TYPE E_Typ_MER_MODE :
(
	/// 0= main mode automatic, controller automatically merge hangers from different lines dependent E_Typ_MER_AUTO_MODE
	Automatic := 0,
	/// 1= main mode on command, in case if merger work as charge controller. Release line X dependent from parent command.
	OnCommand
);
END_TYPE

(* stored: Version 1.1.0.1, ProductVersion 3.1.0.23
   DUT E_Typ_MER_MODE: Id {5c6ff74c-8415-465c-b530-a7a7cb6673b3} *)
